(* CoDeSys 2.3.9.35 project: Q02.pro *)
(* Author: Altus *)
(* Libraries: DU35x.lib 7.7.11 16:00:41, Navigation.lib 15.7.11 10:14:37, SysLibTargetVisu.lib 26.11.08 09:56:12, Standard.lib 26.11.08 09:46:20, Iecsfc.lib 26.11.08 09:46:14, SYSLIBCALLBACK.LIB 26.11.08 09:56:12 *)

(* PLC configuration (modules and I/O channels)
Configuración del PLC [Root] node -1, in %IB0 out %QB0
  Comunicación [Comunica] node 0, in %IB0 out %QB0
    COM1 [COM1] node 0, in %IB0 out %QB0 {BaudRate = 115200; Paridade = No Parity; StopBits = 1 Stop Bit; Modem = Without RTS/CTS; Delay = 5}
      MToolIEC [Codesys] node 0, in %IB0 out %QB0
    COM2 [COM2] node 1, in %IB0 out %QB0 {BaudRate = 115200; Paridade = No Parity; StopBits = 1 Stop Bit; Modem = Without RTS/CTS; Delay = 5}
      Desactivada [Desabilitado485] node 0, in %IB0 out %QB0
  Bus [Barramento] node 1, in %IB0 out %QB0
    Entradas [Entradas] node 0, in %IB0 out %QB0
      Entradas Digitales 0 [Entradas0] node 0, in %IW0 out %QB0
        I00 AT %IX0.0 [BitInput] I0.0
        I01 AT %IX0.1 [BitInput] I0.1
        I02 AT %IX0.2 [BitInput] I0.2
        I03 AT %IX0.3 [BitInput] I0.3
        I04 AT %IX0.4 [BitInput] I0.4
        I05 AT %IX0.5 [BitInput] I0.5
        I06 AT %IX0.6 [BitInput] I0.6
        I07 AT %IX0.7 [BitInput] I0.7
        I08 AT %IX0.8 [BitInput] I0.8
      Entradas Digitales 1 [Entradas1] node 0, in %IW1 out %QB0
        I10 AT %IX1.0 [BitInput] I1.0
        I11 AT %IX1.1 [BitInput] I1.1
        I12 AT %IX1.2 [BitInput] I1.2
        I13 AT %IX1.3 [BitInput] I1.3
        I14 AT %IX1.4 [BitInput] I1.4
        I15 AT %IX1.5 [BitInput] I1.5
        I16 AT %IX1.6 [BitInput] I1.6
        I17 AT %IX1.7 [BitInput] I1.7
        I18 AT %IX1.8 [BitInput] I1.8
      Entradas Digitales 2 [Entradas2] node 0, in %IW2 out %QB0
        I20 AT %IX2.0 [BitInput] I2.0
        I21 AT %IX2.1 [BitInput] I2.1
      Entrada Analógica [EntradaAnalogica] node 0, in %IW4 out %QB0
        AI0 AT %IW4 [WordInput] AI0 {TipoAnalogica = Channel Disable; FiltroAnalogica = Filter 0 - AI=2ms  / AV=90ms; FundoEscala = 0}
        AI1 AT %IW5 [WordInput] AI1 {TipoAnalogica = Channel Disable; FiltroAnalogica = Filter 0 - AI=2ms  / AV=90ms; FundoEscala = 0}
        AI2 AT %IW6 [WordInput] AI2 {TipoAnalogica = Channel Disable; FiltroAnalogica = Filter 0 - AI=2ms  / AV=90ms; FundoEscala = 0}
        AI3 AT %IW7 [WordInput] AI3 {TipoAnalogica = Channel Disable; FiltroAnalogica = Filter 0 - AI=2ms  / AV=90ms; FundoEscala = 0}
      Entradas Rápidas [EntradasRapidas] node 1, in %IB16 out %QB0
        Bloque 0 [Bloco0] node 0, in %IB16 out %QB0
          Desactivado [DesabilitadoBloco0] node 0, in %IB16 out %QB0
        Bloque 1 [Bloco1] node 1, in %IB16 out %QB0
          Desactivado [DesabilitadoBloco1] node 0, in %IB16 out %QB0
        Entrada Configurable Bloque 0 [EntradaConfiBloco0] node 2, in %IB16 out %QB0
          Contador 0 [EntradaConfContador0] node 0, in %IB16 out %QB0 {EntradaConfiguravelContador = Disable}
        Entrada Configurable Bloque 1 [EntradaConfiBloco1] node 3, in %IB16 out %QB0
          Contador 2 [EntradaConfContador2] node 0, in %IB16 out %QB0 {EntradaConfiguravelContador = Disable}
    Salidas [Saidas] node 1, in %IB13 out %QB0
      Salidas Digitales 0 [Saidas0] node 0, in %IW0 out %QW0
        Q00 AT %QX0.0 [BitOutput] Q0.0
        Q01 AT %QX0.1 [BitOutput] Q0.1
        Q02 AT %QX0.2 [BitOutput] Q0.2
        Q03 AT %QX0.3 [BitOutput] Q0.3
        Q04 AT %QX0.4 [BitOutput] Q0.4
        Q05 AT %QX0.5 [BitOutput] Q0.5
        Q06 AT %QX0.6 [BitOutput] Q0.6
        Q07 AT %QX0.7 [BitOutput] Q0.7
      Salidas Digitales 1 [Saidas1] node 0, in %IW0 out %QW1
        Q10 AT %QX1.0 [BitOutput] Q1.0
        Q11 AT %QX1.1 [BitOutput] Q1.1
        Q12 AT %QX1.2 [BitOutput] Q1.2
        Q13 AT %QX1.3 [BitOutput] Q1.3
        Q14 AT %QX1.4 [BitOutput] Q1.4
        Q15 AT %QX1.5 [BitOutput] Q1.5
        Q16 AT %QX1.6 [BitOutput] Q1.6
        Q17 AT %QX1.7 [BitOutput] Q1.7
      Salida Analógica [SaidaAnalogica] node 0, in %IW0 out %QW3
        AO0 AT %QW3 [WordOutput] AO0 {TipoAnalogica = Channel Disable; FundoEscala = 0}
        AO1 AT %QW4 [WordOutput] AO1 {TipoAnalogica = Channel Disable; FundoEscala = 0}
      Salidas Rápidas [SaidasRapidas] node 1, in %IB0 out %QB10
        Salida Rápida 0 Desactivada [DesabilitadoF0] node 0, in %IB0 out %QB10
        Salida Rápida 1 Desactivada [DesabilitadoF1] node 1, in %IB0 out %QB10
      Salidas Común del Contador [SaidasContador] node 2, in %IB0 out %QB10
        Salida del Bloque 0 Desactivada [DesabilitadoSaidaBloco0] node 0, in %IB0 out %QB10
        Salida del Bloque 1 Desactivada [DesabilitadoSaidaBloco1] node 1, in %IB0 out %QB10
  Eventos Externos [Eventos] node 2, in %IB13 out %QB6
    Evento Temporizado [TimerEvent] node 0, in %IB13 out %QB6 {Intervalo = 10}
*)

(* Task configuration *)
TASK MAYOR (PRIORITY := 1, INTERVAL := T#1ms);
	PLC_PRG();
END_TASK
TASK NAVEGACION (PRIORITY := 1, INTERVAL := T#20ms);
	NAVEGACION();
END_TASK
TASK VISUALIZATION (PRIORITY := 1, INTERVAL := T#500ms);
	MAINTARGETVISU_PAINT_CODE();
END_TASK
TASK KEYBOARD_USAGE (PRIORITY := 1, INTERVAL := T#20ms);
	MAINTARGETVISU_INPUT_CODE();
END_TASK

(* POU PLC_PRG, LD *)
PROGRAM PLC_PRG
VAR
END_VAR
VAR_INPUT
	Sensor AT %IX0.0: BOOL;
END_VAR
VAR_OUTPUT
	Valvula AT %QX1.0: BOOL;
	Bomba AT %QX1.1: BOOL;
END_VAR
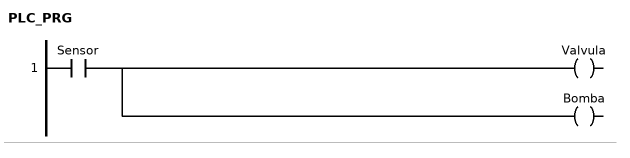
_LD_ (* Ladder Diagram *)
NETWORK 1
	[Sensor] --- (Valvula) (Bomba)
_END_LD_
(* the same logic as Structured Text *)
(* Network 1 *)
Valvula := Sensor;
Bomba := Sensor;
END_PROGRAM

(* POU NAVEGACION, ST *)
PROGRAM NAVEGACION
VAR
	ControleTelas : NAVIGATION;
	ListaTelas 	: ARRAY [0..30] OF STRING(10);
END_VAR
ListaTelas[0] := 'MAIN';

ControleTelas(ENABLE_UPDW := FALSE, VISU_LIST := ListaTelas, UP := FALSE, DOWN := FALSE);
END_PROGRAM
